// TIA Portal V16 export
// export: Created 2022-01-12T14:31:53.9688397Z, ExportSetting WithDefaults, DisplayName Totally Integrated Automation Portal, DisplayVersion V16 Update 4, DisplayName TIA Portal Version Control Interface, DisplayVersion V16 Update 2, DisplayName TIA Portal Openness, DisplayVersion V16 Update 4, DisplayName STEP 7 Professional, DisplayVersion V16 Update 4, DisplayName STEP 7 Safety, DisplayVersion V16, DisplayName WinCC Professional, DisplayVersion V16 Update 4
ORGANIZATION_BLOCK "Main"   // OB1, LAD, ProgramCycle
TITLE = "Main Program Sweep (Cycle)"
{ S7_Optimized_Access := 'TRUE' }
VERSION : 0.1
// stored: AutoNumber true, IsIECCheckEnabled false, SetENOAutomatically false
   VAR_INPUT
      Initial_Call : Bool;   // Initial call of this OB
      Remanence : Bool;   // =True, if remanent data are available
   END_VAR
BEGIN

REGION Network 1 (SCL)
   "ala" := "ala" + 1;
   "obsluga_stacyjki"();
END_REGION

REGION Network 2 (SCL)
   // #dlugosc := INT_TO_WORD(REAL_TO_INT("SIG".SIG[0]));//dlugosc paczki danych
   // //"liznik".liznik > 11 AND "liznik".liznik < 15
   // "BRCV_DB"(EN_R := (1),
   //           ID := W#16#116,
   //           R_ID := 3,
   //           STATUS => "status_reeed",
   //           RD_1 := "SIG".SIG,
   //           LEN := #dlugosc);
   // "R_TRIG_DB"(CLK := ("liznik".liznik >1 AND "liznik".liznik < 3));

   // "BSEND_DB"(REQ := ("R_TRIG_DB".Q),
   //            R := FALSE,
   //            ID := W#16#111,
   //            R_ID := 1,
   //            STATUS => "status_send",
   //            SD_1 := "SIG".SIG,
   //            LEN := #dlugosc);

   //     "PUT_DB"(REQ    := "Clock_10Hz",
   //              ID     := W#16#111,
   //              ADDR_1 := P#DB60.DBX0.0 int 1,
   //              SD_1   := P#DB23.DBX0.0 int 1);
END_REGION
END_ORGANIZATION_BLOCK
